FUNCTION_BLOCK FB_ModeControlBox
VAR_INPUT
END_VAR
VAR_OUTPUT
END_VAR
VAR
END_VAR

END_FUNCTION_BLOCK

(* stored: Version 1.1.0.1, ProductVersion 3.1.4024.10
   POU FB_ModeControlBox: Id {5c8d61b7-c8a3-4bf0-98cd-78798a5dcb40}, SpecialFunc None *)
